(* IEC 61131-3 sources: eCockpitGit/test_project/src/%F%00 Library/%F%Common Functions/%F%Linearsation/%F%INT, 6 files *)

(* ---- %POU%FU_iLinear2.st ---- *)
//This function, converts an x, value to an y value using and 2 points on the x and y scale
// +-----------+----------+----------+-----------------------------------------------------------------------------------------------------------------------+
// |**Version**|**Author**| **Date** |**Changes**                                                                                                            |
// +-----------+----------+----------+-----------------------------------------------------------------------------------------------------------------------+
// | 1         | NSN      | 10-01-18 | Updated to new format                                                                                                 |
// +-----------+----------+----------+-----------------------------------------------------------------------------------------------------------------------+
// | 1.1       | NSN      | 13-06-18 | Updated names and types                                                                                               |
// +-----------+----------+----------+-----------------------------------------------------------------------------------------------------------------------+
FUNCTION FU_iLinear2 : INT
VAR_INPUT
	XIn		:INT;
	X1		:INT;
	X2		:INT;
	Y1		:INT;
	Y2		:INT;
END_VAR
VAR
	a		:REAL;
	b		:REAL;
END_VAR
(*%!%__DELIMITER__%!%*)
IF X2 > X1 THEN
	//a value is calculated
	IF X2 - X1 = 0 THEN	a := 0; ELSE a := TO_REAL((Y2 - Y1)) / (X2 - X1); END_IF
	//b value is calculated
	b 							:=		TO_REAL(Y1) - (a * TO_REAL(X1));
	//Output is calculated
	FU_iLinear2 				:=		TO_INT(a * TO_REAL (XIn) + b);
ELSE
	//a value is calculated
	IF X2 - X1 = 0 THEN	a := 0; ELSE a := TO_REAL((Y2 - Y1)) / (X2 - X1); END_IF
	//b value is calculated
	b 							:=		TO_REAL(Y1) - (a * TO_REAL(X1));
	//Output is calculated
	FU_iLinear2 				:=		TO_INT(a * TO_REAL (XIn) + b);
END_IF

(* ---- %POU%FU_iLinear2Ends.st ---- *)
//This function, converts an x, value to an y value using and 2 points on the x and y scale
//This function has ends, which means the output is never greater or smaller than the range of y
// +-----------+----------+----------+-----------------------------------------------------------------------------------------------------------------------+
// |**Version**|**Author**| **Date** |**Changes**                                                                                                            |
// +-----------+----------+----------+-----------------------------------------------------------------------------------------------------------------------+
// | 1         | NSN      | 03-01-18 | Creation                                                                                                              |
// +-----------+----------+----------+-----------------------------------------------------------------------------------------------------------------------+
// | 1.1       | NSN      | 04-01-18 | Value name changes                                                                                                    |
// +-----------+----------+----------+-----------------------------------------------------------------------------------------------------------------------+
// | 1.2       | NSN      | 13-06-18 | Updated names and types                                                                                               |
// +-----------+----------+----------+-----------------------------------------------------------------------------------------------------------------------+
FUNCTION FU_iLinear2Ends : INT
VAR_INPUT
	XIn		:INT;
	X1		:INT;
	X2		:INT;
	Y1		:INT;
	Y2		:INT;
END_VAR
VAR
	a		:REAL;
	b		:REAL;
END_VAR
(*%!%__DELIMITER__%!%*)
IF X2 > X1 THEN
	IF XIn <= X1 THEN	//When input is out of bounds
		FU_iLinear2Ends 			:=		Y1;
	ELSIF XIn >= X2 THEN	//When input is out of bounds
		FU_iLinear2Ends 			:=		Y2;
	ELSIF XIn > X1 AND XIn < X2 THEN	//When input is with the
		//a value is calculated
		IF X2 - X1 = 0 THEN	a := 0; ELSE a := TO_REAL((Y2 - Y1)) / (X2 - X1); END_IF
		//b value is calculated
		b 							:=		TO_REAL(Y1) - (a * TO_REAL(X1));
		//Output is calculated
		FU_iLinear2Ends 			:=		TO_INT(a * TO_REAL (XIn) + b);
	END_IF
ELSE
	IF XIn >= X1 THEN
		FU_iLinear2Ends 			:=		Y1;
	ELSIF XIn <= X2 THEN
		FU_iLinear2Ends 			:=		Y2;
	ELSIF XIn < X1 AND XIn > X2 THEN
		//a value is calculated
		IF X2 - X1 = 0 THEN	a := 0; ELSE a := TO_REAL((Y2 - Y1)) / (X2 - X1); END_IF
		//b value is calculated
		b 							:=		TO_REAL(Y1) - (a * TO_REAL(X1));
		//Output is calculated
		FU_iLinear2Ends 			:=		TO_INT(a * TO_REAL (XIn) + b);
	END_IF
END_IF

(* ---- %POU%FU_iLinear3Ends.st ---- *)
//This function, converts an x, value to an y value using and 3 points on the x and y scale
//This function has ends, which means the output is never greater or smaller than the range of y
// +-----------+----------+----------+-----------------------------------------------------------------------------------------------------------------------+
// |**Version**|**Author**| **Date** |**Changes**                                                                                                            |
// +-----------+----------+----------+-----------------------------------------------------------------------------------------------------------------------+
// | 1         | NSN      | 10-01-18 | Updated to new format                                                                                                 |
// +-----------+----------+----------+-----------------------------------------------------------------------------------------------------------------------+
// | 1.1       | NSN      | 13-06-18 | Updated names and type                                                                                                |
// +-----------+----------+----------+-----------------------------------------------------------------------------------------------------------------------+
FUNCTION FU_iLinear3Ends : INT
VAR_INPUT
	XIn		:INT;
	X1		:INT;
	X2		:INT;
	X3		:INT;
	Y1		:INT;
	Y2		:INT;
	Y3		:INT;
END_VAR
VAR
	a		:REAL;
	b		:REAL;
END_VAR
(*%!%__DELIMITER__%!%*)
IF X3 > X1 THEN
	IF XIn <= X1 THEN	//When input is out of bounds
		FU_iLinear3Ends 			:=		Y1;
	ELSIF XIn >= X3 THEN	//When input is out of bounds
		FU_iLinear3Ends 			:=		Y3;
	ELSIF XIn > X1 AND XIn <= X2 THEN	//When input is with the
		//a value is calculated
		IF X2 - X1 = 0 THEN	a := 0; ELSE a := TO_REAL((Y2 - Y1)) / (X2 - X1); END_IF
		//b value is calculated
		b 							:=		TO_REAL(Y1) - (a * TO_REAL(X1));
		//Output is calculated
		FU_iLinear3Ends 			:=		TO_INT(a * TO_REAL (XIn) + b);
	ELSIF XIn > X2 AND XIn < X3 THEN
		//a value is calculated
		IF X3 - X2 = 0 THEN	a := 0; ELSE a := TO_REAL((Y3 - Y2)) / (X3 - X2); END_IF
		//b value is calculated
		b 							:=		TO_REAL(Y2) - (a * TO_REAL(X2));
		//Output is calculated
		FU_iLinear3Ends 			:=		TO_INT(a * TO_REAL (XIn) + b);
	END_IF
ELSE
	IF XIn >= X1 THEN
		FU_iLinear3Ends 			:=		Y1;
	ELSIF XIn <= X3 THEN
		FU_iLinear3Ends 			:=		Y3;
	ELSIF XIn < X1 AND XIn >= X2 THEN
		//a value is calculated
		IF X2 - X1 = 0 THEN	a := 0; ELSE a := TO_REAL((Y2 - Y1)) / (X2 - X1); END_IF
		//b value is calculated
		b 							:=		TO_REAL(Y1) - (a * TO_REAL(X1));
		//Output is calculated
		FU_iLinear3Ends 			:=		TO_INT(a * TO_REAL (XIn) + b);
	ELSIF XIn < X2 AND XIn > X3 THEN
		//a value is calculated
		IF X3 - X2 = 0 THEN	a := 0; ELSE a := TO_REAL((Y3 - Y2)) / (X3 - X2); END_IF
		//b value is calculated
		b 							:=		TO_REAL(Y2) - (a * TO_REAL(X2));
		//Output is calculated
		FU_iLinear3Ends 			:=		TO_INT(a * TO_REAL (XIn) + b);
	END_IF
END_IF

(* ---- %POU%FU_iLinear4Ends.st ---- *)
//This function, converts an x, value to an y value using and 3 points on the x and y scale
//This function has ends, which means the output is never greater or smaller than the range of y
// +-----------+----------+----------+-----------------------------------------------------------------------------------------------------------------------+
// |**Version**|**Author**| **Date** |**Changes**                                                                                                            |
// +-----------+----------+----------+-----------------------------------------------------------------------------------------------------------------------+
// | 1         | NSN      | 30-05-18 | Updated to new format                                                                                                 |
// +-----------+----------+----------+-----------------------------------------------------------------------------------------------------------------------+
FUNCTION FU_iLinear4Ends : INT
VAR_INPUT
	XIn		:INT;
	X1		:INT;
	X2		:INT;
	X3		:INT;
	X4		:INT;
	Y1		:INT;
	Y2		:INT;
	Y3		:INT;
	Y4		:INT;
END_VAR
VAR
	a		:REAL;
	b		:REAL;
END_VAR
(*%!%__DELIMITER__%!%*)
IF X4 > X1 THEN
	IF XIn <= X1 THEN	//When input is out of bounds
		FU_iLinear4Ends 			:=		Y1;
	ELSIF XIn >= X4 THEN	//When input is out of bounds
		FU_iLinear4Ends 			:=		Y4;
	ELSIF XIn > X1 AND XIn <= X2 THEN	//When input is with the
		//a value is calculated
		IF X2 - X1 = 0 THEN	a := 0; ELSE a := TO_REAL((Y2 - Y1)) / (X2 - X1); END_IF
		//b value is calculated
		b 							:=		TO_REAL(Y1) - (a * TO_REAL(X1));
		//Output is calculated
		FU_iLinear4Ends 			:=		TO_INT(a * TO_REAL (XIn) + b);
	ELSIF XIn > X2 AND XIn <= X3 THEN
		//a value is calculated
		IF X3 - X2 = 0 THEN	a := 0; ELSE a := TO_REAL((Y3 - Y2)) / (X3 - X2); END_IF
		//b value is calculated
		b 							:=		TO_REAL(Y2) - (a * TO_REAL(X2));
		//Output is calculated
		FU_iLinear4Ends 			:=		TO_INT(a * TO_REAL (XIn) + b);
	ELSIF XIn > X3 AND XIn < X4 THEN
		//a value is calculated
		IF X4 - X3 = 0 THEN	a := 0; ELSE a := TO_REAL((Y4 - Y3)) / (X4 - X3); END_IF
		//b value is calculated
		b 							:=		TO_REAL(Y3) - (a * TO_REAL(X3));
		//Output is calculated
		FU_iLinear4Ends 			:=		TO_INT(a * TO_REAL (XIn) + b);
	END_IF
ELSE
	IF XIn >= X1 THEN
		FU_iLinear4Ends 			:=		Y1;
	ELSIF XIn <= X4 THEN
		FU_iLinear4Ends 			:=		Y4;
	ELSIF XIn < X1 AND XIn >= X2 THEN
		//a value is calculated
		IF X2 - X1 = 0 THEN	a := 0; ELSE a := TO_REAL((Y2 - Y1)) / (X2 - X1); END_IF
		//b value is calculated
		b 							:=		TO_REAL(Y1) - (a * TO_REAL(X1));
		//Output is calculated
		FU_iLinear4Ends 			:=		TO_INT(a * TO_REAL (XIn) + b);
	ELSIF XIn < X2 AND XIn >= X3 THEN
		//a value is calculated
		IF X3 - X2 = 0 THEN	a := 0; ELSE a := TO_REAL((Y3 - Y2)) / (X3 - X2); END_IF
		//b value is calculated
		b 							:=		TO_REAL(Y2) - (a * TO_REAL(X2));
		//Output is calculated
		FU_iLinear4Ends 			:=		TO_INT(a * TO_REAL (XIn) + b);
	ELSIF XIn < X3 AND XIn > X4 THEN
		//a value is calculated
		IF X4 - X3 = 0 THEN	a := 0; ELSE a := TO_REAL((Y4 - Y3)) / (X4 - X3); END_IF
		//b value is calculated
		b 							:=		TO_REAL(Y3) - (a * TO_REAL(X3));
		//Output is calculated
		FU_iLinear4Ends 			:=		TO_INT(a * TO_REAL (XIn) + b);
	END_IF
END_IF

(* ---- %POU%FU_iLinearXEnds.st ---- *)
//This function, converts an x, value to an y value using and x amount of points on the x and y scale
//This function has ends, which means the output is never greater or smaller than the range of y
// +-----------+----------+----------+-----------------------------------------------------------------------------------------------------------------------+
// |**Version**|**Author**| **Date** |**Changes**                                                                                                            |
// +-----------+----------+----------+-----------------------------------------------------------------------------------------------------------------------+
// | 1         | NSN      | 03-01-18 | Creation                                                                                                              |
// +-----------+----------+----------+-----------------------------------------------------------------------------------------------------------------------+
FUNCTION FU_iLinearXEnds : INT
VAR_INPUT
	iXIn		:INT;				//Input value to be linearised
	pXArray		:POINTER TO INT;	//Address of x array
	pYArray		:POINTER TO INT; 	//Address of y array
	uiSize		:UINT;				//Amount of points in
END_VAR
VAR
	LowerLimit	:BOOL;
	UpperLimit	:BOOL;
	UpperXAdr	:POINTER TO INT;	//Buffer for current x address
	LowerXAdr	:POINTER TO INT;	//Buffer for current x address
	UpperYAdr	:POINTER TO INT; 	//Buffer for current y address
	LowerYAdr	:POINTER TO INT; 	//Buffer for current y address
	FOR1		:UINT;
	a			:REAL;
	b			:REAL;
	d			:BOOL;
END_VAR
(*%!%__DELIMITER__%!%*)
IF uiSize > 1 THEN
	//Direction is found
	UpperXAdr					:=		pXArray + 2;
	d							:=		UpperXAdr^ > pXArray^;

	//Pointers are set
	UpperXAdr					:=		pXArray;
	UpperYAdr					:=		pYArray;

	FOR FOR1 := 1 TO uiSize DO
		IF d THEN
			IF UpperXAdr^ <= iXIn THEN
				IF FOR1 = uiSize AND UpperXAdr^ <> iXIn THEN
					UpperLimit	:=		TRUE;
				ELSIF FOR1 <> uiSize THEN
					UpperXAdr	:=		UpperXAdr + 2;
					UpperYAdr	:=		UpperYAdr + 2;
				END_IF
			ELSE
				IF pXArray = UpperXAdr THEN
					LowerLimit	:=		TRUE;
				ELSE
					LowerXAdr	:=		UpperXAdr - 2;
					LowerYAdr	:=		UpperYAdr - 2;
				END_IF
				Exit;
			END_IF
		ELSE
			IF UpperXAdr^ >= iXIn THEN
				IF FOR1 = uiSize AND UpperXAdr^ <> iXIn THEN
					UpperLimit	:=		TRUE;
				ELSIF FOR1 <> uiSize THEN
					UpperXAdr	:=		UpperXAdr + 2;
					UpperYAdr	:=		UpperYAdr + 2;
				END_IF
			ELSE
				IF pXArray = UpperXAdr THEN
					LowerLimit	:=		TRUE;
				ELSE
					LowerXAdr	:=		UpperXAdr - 2;
					LowerYAdr	:=		UpperYAdr - 2;
				END_IF
				Exit;
			END_IF
		END_IF
	END_FOR

	IF LowerLimit THEN
		FU_iLinearXEnds				:=		pYArray^;
	ELSIF UpperLimit THEN
		FU_iLinearXEnds				:=		UpperYAdr^;
	ELSE
		IF iXIn = UpperXAdr^ THEN
			FU_iLinearXEnds			:=		UpperYAdr^;
		ELSIF iXIn = LowerXAdr^ THEN
			FU_iLinearXEnds			:=		LowerYAdr^;
		ELSE
			IF UpperXAdr^ - LowerXAdr^ = 0 THEN
				a				:=		0;
			ELSE
				a				:=		TO_REAL(UpperYAdr^ - LowerYAdr^) / TO_REAL(UpperXAdr^ - LowerXAdr^);
			END_IF
			b					:=		TO_REAL(LowerYAdr^) - (a * TO_REAL(LowerXAdr^));
			FU_iLinearXEnds 		:=		TO_INT(a * TO_REAL(iXIn) + b);
		END_IF
	END_IF
END_IF

(* ---- %POU%FU_iLinearXFixed.st ---- *)
//This function, converts an x value to a fixed y value
//When the input is between two x values, the corresponding y value is outputted
// +-----------+----------+----------+-----------------------------------------------------------------------------------------------------------------------+
// |**Version**|**Author**| **Date** |**Changes**                                                                                                            |
// +-----------+----------+----------+-----------------------------------------------------------------------------------------------------------------------+
// | 1         | NSN      | 03-01-18 | Creation                                                                                                              |
// +-----------+----------+----------+-----------------------------------------------------------------------------------------------------------------------+
// | 1.1       | NSN      | 13-06-18 | Updated names and types                                                                                               |
// +-----------+----------+----------+-----------------------------------------------------------------------------------------------------------------------+
FUNCTION FU_iLinearXFixed : INT
VAR_INPUT
	iXIn		:INT;					//Input value
	pXArray		:POINTER TO INT;		//Address of x array
	uiXSize		:UINT;					//Size of x array
	pYArray		:POINTER TO INT; 		//Address of y array
	uiYSize		:UINT; 					//Size of y array
END_VAR
VAR
	XAddBuff	:POINTER TO INT;
	SmallestSize:UINT;
END_VAR
(*%!%__DELIMITER__%!%*)
XAddBuff				:=		pXArray + 2;
IF uiXSize > uiYSize THEN
	SmallestSize		:=		uiYSize;
ELSE
	SmallestSize		:=		uiXSize;
END_IF
IF pXArray^ < XAddBuff^ THEN
	WHILE SmallestSize > 0 DO
		SmallestSize			:=		SmallestSize - 1;
		IF iXIn < XAddBuff^ OR SmallestSize = 0 THEN
			FU_iLinearXFixed	:=		pYArray^;
			RETURN;
		ELSE
			XAddBuff			:=		XAddBuff + 2;
			pYArray				:=		pYArray + 2;
		END_IF
	END_WHILE
ELSE
	WHILE SmallestSize > 0 DO
		SmallestSize			:=		SmallestSize - 1;
		IF iXIn > XAddBuff^ OR SmallestSize = 0 THEN
			FU_iLinearXFixed	:=		pYArray^;
			RETURN;
		ELSE
			XAddBuff			:=		XAddBuff + 2;
			pYArray				:=		pYArray + 2;
		END_IF
	END_WHILE
END_IF
